// TIA Portal V17 export
// export: Created 2024-08-09T12:53:15.4005654Z, ExportSetting WithDefaults, DisplayName Totally Integrated Automation Portal, DisplayVersion V17 Update 7, DisplayName TIA Portal Openness, DisplayVersion V17 Update 7, DisplayName TIA Portal Version Control Interface, DisplayVersion V17, DisplayName STEP 7 Professional, DisplayVersion V17 Update 7, DisplayName STEP 7 Safety, DisplayVersion V17 Update 6, DisplayName WinCC Professional, DisplayVersion V17 Update 7
VAR_GLOBAL   // PLC tag table "Dec_Niveaux_GTOUR"
END_VAR
VAR_GLOBAL CONSTANT   // user constants
   NIV_GTOUR_DEM_CHARG : USInt := 10;
END_VAR
